// TwinCAT 3 PLC project TcPrpNodeTableSample
// ProgramVersion: 3.1.4026.10
// libraries:
//   Tc2_Standard, * (Beckhoff Automation GmbH)
//   Tc2_System, * (Beckhoff Automation GmbH)
//   Tc3_Module, * (Beckhoff Automation GmbH)
// project tree:
//   DUTs/ STcPrpLinkStatus.TcDUT (not stored), STcPrpNodeEntry.TcDUT
//   GVLs/ VAR_OIDs.TcGVL (not stored)
//   / PlcTask.TcTTO
//   POUs/ FB_TcPrpAdapter.TcPOU, FB_TcPrpNode.TcPOU, MAIN.TcPOU
// real-time tasks:
//   TASK PlcTask: cycle T#10ms, priority 20, ADS port 350
// I/O:
//   DEVICE X000 (RT-Ethernet Adapter)
//   DEVICE X001 (RT-Ethernet Adapter)

CONFIGURATION TcPrpNodeTableSample
    RESOURCE PLC ON TwinCAT3
        TASK PlcTask(INTERVAL := T#10ms, PRIORITY := 20);
        PROGRAM MAIN WITH PlcTask : MAIN;
    END_RESOURCE
END_CONFIGURATION

// ---- DUTs/STcPrpNodeEntry.TcDUT
TYPE STcPrpNodeEntry : 
STRUCT
	(* MAC Address of the remote source node. *)
	{attribute 'GUID' := 'CC07E0A0-FC03-45CD-BFD9-D46B7C731E7B'}
	MacAddress : MAC_ADDRESS;
	(* True if the node is probably a SAN on port A. *)
	bSanA : BOOL;
	(* True if the node is probably a SAN on port B. *)
	bSanB : BOOL;
	(* Number of frames received from that node on port A. *)
	CntReceivedA : UDINT;
	(* Number of frames received from that node on port B. *)
	CntReceivedB : UDINT;
	(* Number of frames received from that node with wrong LAN identifier on port A. *)
	CntErrWrongLanA : UDINT;
	(* Number of frames received from that node with wrong LAN identifier on port B. *)
	CntErrWrongLanB : UDINT;
	(* Discarded dublicated frames count fron node on port A. *)
	CntDuplicateDiscardLanA : UDINT;
	(* Discarded dublicated frames count fron node on port B. *)
	CntDuplicateDiscardLanB : UDINT;
	(* Supervision frames count from node on port A. *)
	CntSupervisionFrameLanA : UDINT;
	(* Supervision frames count from node on port B. *)
	CntSupervisionFrameLanB : UDINT;
	(* Receive error count from node on port A. *)
	CntRxErrLanA : UDINT;
	(* Receive error count from node on port B. *)
	CntRxErrLanB : UDINT;
	(* Transmit error count from node on port A. *)
	CntTxErrLanA : UDINT;
	(* Transmit error count from node on port B. *)
	CntTxErrLanB : UDINT;
	(* Time at which the latest frame was received from that node over port A. *)
	TimeLastSeenA : UDINT;
	(* Time at which the latest frame was received from that node over port B. *)
	TimeLastSeenB : UDINT;
END_STRUCT
END_TYPE

// ---- POUs/MAIN.TcPOU
PROGRAM MAIN
VAR
	fbAdapter : FB_TcPrpAdapter(VAR_OIDs.PRP);
	fbNode : FB_TcPrpNode(MAC);
END_VAR
VAR CONSTANT
	MAC : MAC_ADDRESS := ( b := [16#00, 16#01, 16#05, 16#62, 16#42, 16#F5] );
END_VAR

fbNode(fbAdapter:= fbAdapter);
fbNode.bTimeoutA; 
fbNode.bTimeoutB; 
fbNode.bDisconnect; 
fbNode.bDisconnected;

END_PROGRAM

// ---- POUs/FB_TcPrpAdapter.TcPOU
FUNCTION_BLOCK PUBLIC FB_TcPrpAdapter
VAR_OUTPUT
	bLinkA : BOOL;
	bLinkB : BOOL;
END_VAR
VAR
	_bValid : BOOL;
	_hResult : HRESULT;
	_nObjectID : OTCID;
	_ipObject : ITComObject;
	_mLinkStatus : STcPrpLinkStatus;
	_nNodeCount : UDINT;
	_arrNodeTable : ARRAY[1.._nNodeTableSize] OF STcPrpNodeEntry;
	_fbAdsRead : ADSREAD;
END_VAR
VAR CONSTANT
	_nNodeTableSize : UDINT := 64;
END_VAR

METHOD FB_exit : BOOL
VAR_INPUT
	bInCopyCode : BOOL; // if TRUE, the exit method is called for exiting an instance that is copied afterwards (online change).
END_VAR
IF bInCopyCode THEN RETURN; END_IF

_bValid := FALSE;

FW_SafeRelease(ADR(_ipObject));
END_METHOD

METHOD FB_init : BOOL
VAR_INPUT
	bInitRetains : BOOL; // if TRUE, the retain variables are initialized (warm start / cold start)
	bInCopyCode : BOOL;  // if TRUE, the instance afterwards gets moved into the copy code (online change)
	
	OID : OTCID; // ObjectID of the PRP Adapter
END_VAR
IF bInCopyCode THEN RETURN; END_IF

_nObjectID := OID;

_hResult := FW_ObjMgr_GetObjectInstance(
	oid:= _nObjectID,
	iid:= TC_GLOBAL_IID_LIST.IID_ITComObject,
	pipUnk:= ADR(_ipObject));

_bValid := SUCCEEDED(_hResult);
END_METHOD

METHOD PUBLIC GetLinkStatus : BOOL
GetLinkStatus := GetObjPara(16#03150005, SIZEOF(_mLinkStatus), ADR(_mLinkStatus));

IF NOT GetLinkStatus THEN
	_mLinkStatus.bLinkA := FALSE;
	_mLinkStatus.bLinkB := FALSE;
END_IF
END_METHOD

METHOD PUBLIC GetNodeCount : UDINT
IF GetObjPara(16#0315000A, SIZEOF(_nNodeCount), ADR(_nNodeCount)) THEN
	GetNodeCount := _nNodeCount;
END_IF
END_METHOD

METHOD PUBLIC GetNodeEntry : BOOL
VAR_INPUT
	nIndex : UDINT;
END_VAR
VAR_IN_OUT
	mEntry : STcPrpNodeEntry;
END_VAR
IF _nNodeCount = 0 THEN
	GetNodeCount();
END_IF
IF _nNodeCount >= _nNodeTableSize THEN
	_nNodeCount := _nNodeTableSize;
END_IF

IF nIndex >= 1 AND nIndex <= _nNodeCount THEN
	mEntry := _arrNodeTable[nIndex];
	GetNodeEntry := TRUE;
END_IF
END_METHOD

METHOD PUBLIC GetNodeIndexByMac : UDINT
VAR_INPUT
	mMacAddress : MAC_ADDRESS;
END_VAR
VAR
	_nIndex : UDINT;
END_VAR
IF _nNodeCount = 0 THEN
	GetNodeCount();
END_IF
IF _nNodeCount >= _nNodeTableSize THEN
	_nNodeCount := _nNodeTableSize;
END_IF

FOR _nIndex := 1 TO _nNodeCount DO
	IF MEMCMP(ADR(_arrNodeTable[_nIndex].MacAddress), ADR(mMacAddress), SIZEOF(mMacAddress)) = 0 THEN
		GetNodeIndexByMac := _nIndex;
		RETURN;
	END_IF
END_FOR
END_METHOD

METHOD PUBLIC GetNodeTable : BOOL
IF NOT _fbAdsRead.BUSY THEN
	_fbAdsRead(READ := FALSE);
END_IF

_fbAdsRead(
	READ:= TRUE,
	PORT:= 10,
	IDXGRP:= _nObjectID,
	IDXOFFS:= 16#03150004,
	LEN:= SIZEOF(_arrNodeTable), 
	DESTADDR:= ADR(_arrNodeTable));

IF _fbAdsRead.ERR THEN
	_hResult := UDINT_TO_DINT(16#98110000 + _fbAdsRead.ERRID);
END_IF

GetNodeTable := NOT (_fbAdsRead.BUSY OR _fbAdsRead.ERR);
END_METHOD

METHOD INTERNAL GetObjPara : BOOL
VAR_INPUT
	nPID : PTCID;
	nData : UDINT;
	pData : PVOID;
END_VAR
IF NOT _bValid THEN RETURN; END_IF

_hResult := _ipObject.TcGetObjPara(nPID, nData, pData, 0);

GetObjPara := SUCCEEDED(_hResult);
END_METHOD

PROPERTY PUBLIC IsValid : BOOL
GET
IsValid := _bValid;
END_GET
END_PROPERTY

PROPERTY PUBLIC LinkStatusA : BOOL
GET
LinkStatusA := _mLinkStatus.bLinkA;
END_GET
END_PROPERTY

PROPERTY PUBLIC LinkStatusB : BOOL
GET
LinkStatusB := _mLinkStatus.bLinkB;
END_GET
END_PROPERTY

PROPERTY Result : HRESULT
GET
Result := _hResult;
END_GET
END_PROPERTY

END_FUNCTION_BLOCK

// ---- POUs/FB_TcPrpNode.TcPOU
FUNCTION_BLOCK FB_TcPrpNode
VAR_IN_OUT
	fbAdapter : FB_TcPrpAdapter;
END_VAR
VAR_OUTPUT
	bValid : BOOL;
	bSan : BOOL; // singly attached node
	bError : BOOL; // any error
	bErrRx : BOOL; // receive errors
	bErrTx : BOOL; // transmit errors
	bErrWrongLan : BOOL; // node with wrong LAN identifier
	bReceived : BOOL; // anything received
	bReceivedA : BOOL; // anything received on adapter A
	bReceivedB : BOOL; // anything received on adapter B
	bTimeoutA : BOOL; // nothing received on adapter A over 2s
	bTimeoutB : BOOL; // nothing received on adapter B over 2s
	bDisconnect : BOOL; // nothing received over 5s
	bDisconnected : BOOL; // nothing received over 5s once
END_VAR
VAR
	_mMacAddress : MAC_ADDRESS;

	_nNodeIndex : UDINT := 16#FFFFFFFF;
	_nNodeCount : UDINT;
	_nNodeCountLast : UDINT;
	_mNodeEntry : STcPrpNodeEntry;
	_mNodeLast : STcPrpNodeEntry;
	
	_bReceiveA : BOOL;
	_bReceiveB : BOOL;
	_bDiscardA :BOOL;
	_bDiscardB : BOOL;
	_bSupervisionA : BOOL;
	_bSupervisionB : BOOL;
	
	_tTimeoutA : TON;
	_tTimeoutB : TON;
	_tDisconnect : TON;
END_VAR
VAR CONSTANT
	ctTimeout : TIME := T#2S;
END_VAR

bReceived := FALSE;
bReceivedA := FALSE;
bReceivedB := FALSE;

IF fbAdapter.IsValid THEN
	_nNodeCount := fbAdapter.GetNodeCount();
	IF fbAdapter.GetNodeTable() THEN
		// get node index if undefined or node count has changed
		IF _nNodeIndex = 16#FFFFFFFF OR _nNodeCount <> _nNodeCountLast THEN
			_nNodeIndex := fbAdapter.GetNodeIndexByMac(_mMacAddress);
			_nNodeCountLast := _nNodeCount;
		END_IF
		// get node entry by index
		bValid := fbAdapter.GetNodeEntry(_nNodeIndex, _mNodeEntry);
		// get node index if  index has changed, inidcated if mac is not as expected			
		IF MEMCMP(ADR(_mNodeEntry.MacAddress), ADR(_mMacAddress), SIZEOF(_mMacAddress)) <> 0 THEN
			_nNodeIndex := fbAdapter.GetNodeIndexByMac(_mMacAddress);	
			bValid := fbAdapter.GetNodeEntry(_nNodeIndex, _mNodeEntry);			
		END_IF

		IF bValid THEN
			bSan := _mNodeEntry.bSanA OR _mNodeEntry.bSanB;
			
			CntError(bErrRx, _mNodeEntry.CntRxErrLanA, _mNodeLast.CntRxErrLanA);
			CntError(bErrRx, _mNodeEntry.CntRxErrLanB, _mNodeLast.CntRxErrLanB);
			
			CntError(bErrTx, _mNodeEntry.CntTxErrLanA, _mNodeLast.CntTxErrLanA);
			CntError(bErrTx, _mNodeEntry.CntTxErrLanB, _mNodeLast.CntTxErrLanB);
	
			CntError(bErrWrongLan, _mNodeEntry.CntErrWrongLanA, _mNodeLast.CntErrWrongLanA);
			CntError(bErrWrongLan, _mNodeEntry.CntErrWrongLanB, _mNodeLast.CntErrWrongLanB);
	
			bError := bErrRx OR bErrTx OR bErrWrongLan;
	
			CntCheck(_bReceiveA, _mNodeEntry.CntReceivedA, _mNodeLast.CntReceivedA);
			CntCheck(_bReceiveB, _mNodeEntry.CntReceivedB, _mNodeLast.CntReceivedB);
	
			CntCheck(_bDiscardA, _mNodeEntry.CntDuplicateDiscardLanA, _mNodeLast.CntDuplicateDiscardLanA);
			CntCheck(_bDiscardB, _mNodeEntry.CntDuplicateDiscardLanB, _mNodeLast.CntDuplicateDiscardLanB);
	
			CntCheck(_bSupervisionA, _mNodeEntry.CntSupervisionFrameLanA, _mNodeLast.CntSupervisionFrameLanA);
			CntCheck(_bSupervisionB, _mNodeEntry.CntSupervisionFrameLanB, _mNodeLast.CntSupervisionFrameLanB);
	
			bReceivedA := _bReceiveA OR _bDiscardA OR _bSupervisionA;
			bReceivedB := _bReceiveB OR _bDiscardB OR _bSupervisionB;
			bReceived := bReceivedA OR bReceivedB;
		END_IF
	END_IF
END_IF

_tTimeoutA(IN := NOT bReceivedA, PT := ctTimeout, Q => bTimeoutA);
_tTimeoutB(IN := NOT bReceivedB, PT := ctTimeout, Q => bTimeoutB);
_tDisconnect(IN := NOT bReceived, PT := T#5S, Q => bDisconnect);
IF bDisconnect THEN bDisconnected := TRUE; END_IF

METHOD PRIVATE CntCheck : BOOL
VAR_IN_OUT
	bChk : BOOL;
	nCnt : UDINT;
	nLst : UDINT;
END_VAR
bChk := nCnt <> nLst;
nLst := nCnt;
END_METHOD

METHOD PRIVATE CntError : BOOL
VAR_IN_OUT
	bErr : BOOL;
	nCnt : UDINT;
	nLst : UDINT;
END_VAR
IF nCnt <> nLst THEN
	bErr := TRUE;
	nLst := nCnt;
END_IF
END_METHOD

METHOD FB_Init : BOOL
VAR_INPUT
	bInitRetains : BOOL; // if TRUE, the retain variables are initialized (warm start / cold start)
	bInCopyCode : BOOL;  // if TRUE, the instance afterwards gets moved into the copy code (online change)
	
	MacAddress : MAC_ADDRESS;
END_VAR
_mMacAddress := MacAddress;
END_METHOD

PROPERTY PUBLIC IsValid : BOOL
GET
IsValid := bValid;
END_GET
END_PROPERTY

METHOD Reset : BOOL
_mNodeLast := _mNodeEntry;

_tTimeoutA(IN := FALSE);
_tTimeoutB(IN := FALSE);
_tDisconnect(IN := FALSE);

bErrRx := FALSE;
bErrTx := FALSE;
bErrWrongLan := FALSE;

bTimeoutA := FALSE;
bTimeoutB := FALSE;
bDisconnect := FALSE;
bDisconnected := FALSE;
END_METHOD

END_FUNCTION_BLOCK
